# EPICS substitutions: db/plsci.substitutions
# P is supplied by dbLoadTemplate() in st.cmd.
file "db/tof.template"
{
    pattern
    {
        CHAMBER,PMT
    }

# FPF2		1	6	 x86l-208
# FPF4		2	6	 x86l-209
# FMF1		3	6	 x86l-209
# FMF2		4	8	x86l-132/212
# FMF3		5	6	x86l-132/212
# FHF1		6	8	x86l-132/212

    { FMF2,1 }
    { FMF2,2 }
    { FMF2,3 }
    { FMF2,4 }
    { FMF2,5 }
    { FMF2,6 }
    { FMF2,7 }
    { FMF2,8 }

    { FHF1,1 }
    { FHF1,2 }
    { FHF1,3 }
    { FHF1,4 }
    { FHF1,5 }
    { FHF1,6 }
    { FHF1,7 }
    { FHF1,8 }
}
